// TIA Portal V20 export
// export: Created 2025-12-01T14:57:27.0785066Z, ExportSetting None, DisplayName Totally Integrated Automation Portal, DisplayVersion V20 Update 3, DisplayName TIA Portal Openness, DisplayVersion V20 Update 3, DisplayName TIA Portal Version Control Interface, DisplayVersion V20 Update 3, DisplayName STEP 7 Professional, DisplayVersion V20 Update 3, DisplayName STEP 7 Safety, DisplayVersion V20 Update 2, DisplayName WinCC Basic/Comfort/Advanced, DisplayVersion V20 Update 3, DisplayName WinCC Professional, DisplayVersion V20 Update 3, DisplayName WinCC Unified, DisplayVersion V20 Update 3
FUNCTION_BLOCK "FB609_RepartoEntradas_2E_Quimarox"   // FB609, LAD
{ S7_Optimized_Access := 'FALSE' }
// stored: AutoNumber false, SetENOAutomatically false
   VAR_INPUT
      Mesa_E1 : UInt;
      Mesa_E2 : UInt;
      AVTF_ME1_MSig : Bool;
      AVTF_ME2_MSig : Bool;
      V_Reparto_ME1 : UInt;
      V_Reparto_ME2 : UInt;
   END_VAR
   VAR_OUTPUT
      Permiso_ME1_MSig : Bool;
      Permiso_ME2_MSig : Bool;
   END_VAR
   VAR
      CNT_Entradas_ME1 : UInt;
      CNT_Entradas_ME2 : UInt;
      MFP_Entrada_ME1 : Bool;
      MFP_Entrada_ME2 : Bool;
      MEntrando_ME1 : Bool;
      MEntrando_ME2 : Bool;
   END_VAR
   VAR_TEMP   // added for the SCL form of the ladder/FBD networks
      _w1 : Bool;
   END_VAR
BEGIN

REGION Network 1: >>>>>>>> INICIALIZAR
END_REGION

REGION Network 2: >>>>>>>> CONTROL DE LOS CONTADORES DE LAS ENTRADAS
END_REGION

REGION Network 3: Numero de Entradas realizadas desde ME1 (Contador)
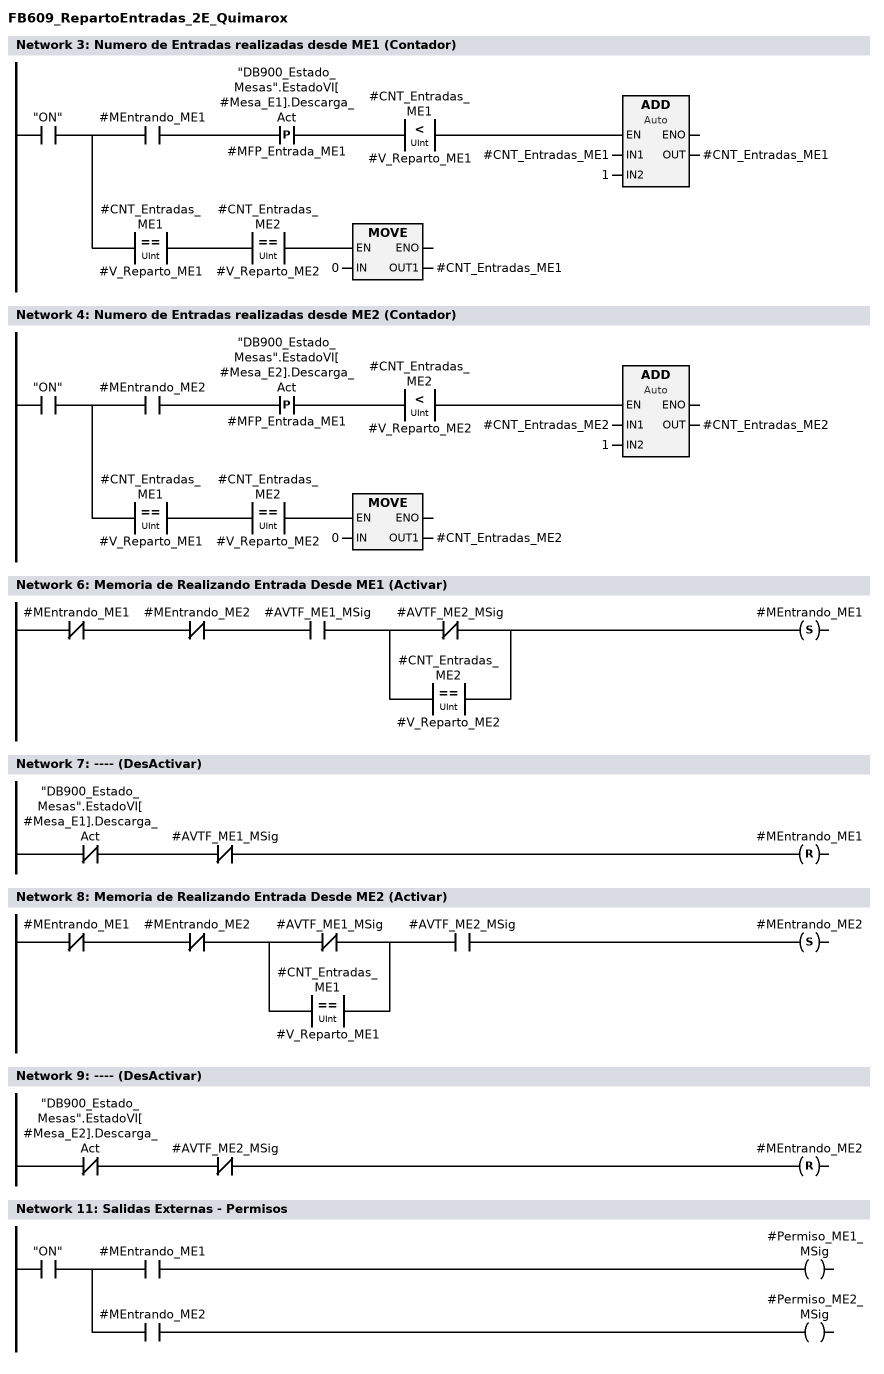
   RUNG wire#powerrail
      Contact( "ON" )
      wire#w1
      Contact( #MEntrando_ME1 )
      P_Contact(operand := "DB900_Estado_Mesas".EstadoVI[#Mesa_E1].Descarga_Act, bit := #MFP_Entrada_ME1)
      { S7_Templates := "SrcType := UInt" } LT_Contact(in1 := #CNT_Entradas_ME1, in2 := #V_Reparto_ME1)
      Add(in1 := #CNT_Entradas_ME1, in2 := 1, out => #CNT_Entradas_ME1)
   END_RUNG
   RUNG wire#w1
      { S7_Templates := "SrcType := UInt" } EQ_Contact(in1 := #CNT_Entradas_ME1, in2 := #V_Reparto_ME1)
      { S7_Templates := "SrcType := UInt" } EQ_Contact(in1 := #CNT_Entradas_ME2, in2 := #V_Reparto_ME2)
      Move(in := 0, out1 => #CNT_Entradas_ME1)
   END_RUNG
   // the same network as SCL:
   #_w1 := "ON" AND #MEntrando_ME1 AND "DB900_Estado_Mesas".EstadoVI[#Mesa_E1].Descarga_Act AND NOT #MFP_Entrada_ME1;   // rising edge of "DB900_Estado_Mesas".EstadoVI[#Mesa_E1].Descarga_Act
   #MFP_Entrada_ME1 := "DB900_Estado_Mesas".EstadoVI[#Mesa_E1].Descarga_Act;
   IF #_w1 AND (#CNT_Entradas_ME1 < #V_Reparto_ME1) THEN #CNT_Entradas_ME1 := #CNT_Entradas_ME1 + 1; END_IF;
   IF "ON" AND (#CNT_Entradas_ME1 = #V_Reparto_ME1) AND (#CNT_Entradas_ME2 = #V_Reparto_ME2) THEN
       #CNT_Entradas_ME1 := 0;
   END_IF;
END_REGION

REGION Network 4: Numero de Entradas realizadas desde ME2 (Contador)
   RUNG wire#powerrail
      Contact( "ON" )
      wire#w1
      Contact( #MEntrando_ME2 )
      P_Contact(operand := "DB900_Estado_Mesas".EstadoVI[#Mesa_E2].Descarga_Act, bit := #MFP_Entrada_ME1)
      { S7_Templates := "SrcType := UInt" } LT_Contact(in1 := #CNT_Entradas_ME2, in2 := #V_Reparto_ME2)
      Add(in1 := #CNT_Entradas_ME2, in2 := 1, out => #CNT_Entradas_ME2)
   END_RUNG
   RUNG wire#w1
      { S7_Templates := "SrcType := UInt" } EQ_Contact(in1 := #CNT_Entradas_ME1, in2 := #V_Reparto_ME1)
      { S7_Templates := "SrcType := UInt" } EQ_Contact(in1 := #CNT_Entradas_ME2, in2 := #V_Reparto_ME2)
      Move(in := 0, out1 => #CNT_Entradas_ME2)
   END_RUNG
   // the same network as SCL:
   #_w1 := "ON" AND #MEntrando_ME2 AND "DB900_Estado_Mesas".EstadoVI[#Mesa_E2].Descarga_Act AND NOT #MFP_Entrada_ME1;   // rising edge of "DB900_Estado_Mesas".EstadoVI[#Mesa_E2].Descarga_Act
   #MFP_Entrada_ME1 := "DB900_Estado_Mesas".EstadoVI[#Mesa_E2].Descarga_Act;
   IF #_w1 AND (#CNT_Entradas_ME2 < #V_Reparto_ME2) THEN #CNT_Entradas_ME2 := #CNT_Entradas_ME2 + 1; END_IF;
   IF "ON" AND (#CNT_Entradas_ME1 = #V_Reparto_ME1) AND (#CNT_Entradas_ME2 = #V_Reparto_ME2) THEN
       #CNT_Entradas_ME2 := 0;
   END_IF;
END_REGION

REGION Network 5: >>>>>>>> MEMORIA DE ESTADO - ENTRANDO
END_REGION

REGION Network 6: Memoria de Realizando Entrada Desde ME1 (Activar)
   RUNG wire#powerrail
      I_Contact( #MEntrando_ME1 )
      I_Contact( #MEntrando_ME2 )
      Contact( #AVTF_ME1_MSig )
      wire#w1
      I_Contact( #AVTF_ME2_MSig )
      wire#w2
      S_Coil( #MEntrando_ME1 )
   END_RUNG
   RUNG wire#w1
      { S7_Templates := "SrcType := UInt" } EQ_Contact(in1 := #CNT_Entradas_ME2, in2 := #V_Reparto_ME2)
   END_RUNG wire#w2
   // the same network as SCL:
   IF NOT #MEntrando_ME1 AND NOT #MEntrando_ME2 AND #AVTF_ME1_MSig AND (NOT #AVTF_ME2_MSig OR (#CNT_Entradas_ME2 = #V_Reparto_ME2)) THEN
       #MEntrando_ME1 := TRUE;
   END_IF;
END_REGION

REGION Network 7: ---- (DesActivar)
   RUNG wire#powerrail
      I_Contact( "DB900_Estado_Mesas".EstadoVI[#Mesa_E1].Descarga_Act )
      I_Contact( #AVTF_ME1_MSig )
      R_Coil( #MEntrando_ME1 )
   END_RUNG
   // the same network as SCL:
   IF NOT "DB900_Estado_Mesas".EstadoVI[#Mesa_E1].Descarga_Act AND NOT #AVTF_ME1_MSig THEN
       #MEntrando_ME1 := FALSE;
   END_IF;
END_REGION

REGION Network 8: Memoria de Realizando Entrada Desde ME2 (Activar)
   RUNG wire#powerrail
      I_Contact( #MEntrando_ME1 )
      I_Contact( #MEntrando_ME2 )
      wire#w1
      I_Contact( #AVTF_ME1_MSig )
      wire#w2
      Contact( #AVTF_ME2_MSig )
      S_Coil( #MEntrando_ME2 )
   END_RUNG
   RUNG wire#w1
      { S7_Templates := "SrcType := UInt" } EQ_Contact(in1 := #CNT_Entradas_ME1, in2 := #V_Reparto_ME1)
   END_RUNG wire#w2
   // the same network as SCL:
   IF NOT #MEntrando_ME1 AND NOT #MEntrando_ME2 AND (NOT #AVTF_ME1_MSig OR (#CNT_Entradas_ME1 = #V_Reparto_ME1)) AND #AVTF_ME2_MSig THEN
       #MEntrando_ME2 := TRUE;
   END_IF;
END_REGION

REGION Network 9: ---- (DesActivar)
   RUNG wire#powerrail
      I_Contact( "DB900_Estado_Mesas".EstadoVI[#Mesa_E2].Descarga_Act )
      I_Contact( #AVTF_ME2_MSig )
      R_Coil( #MEntrando_ME2 )
   END_RUNG
   // the same network as SCL:
   IF NOT "DB900_Estado_Mesas".EstadoVI[#Mesa_E2].Descarga_Act AND NOT #AVTF_ME2_MSig THEN
       #MEntrando_ME2 := FALSE;
   END_IF;
END_REGION

REGION Network 10: >>>>>>>> ACTIVACION DE SALIDAS
END_REGION

REGION Network 11: Salidas Externas - Permisos
   RUNG wire#powerrail
      Contact( "ON" )
      wire#w1
      Contact( #MEntrando_ME1 )
      Coil( #Permiso_ME1_MSig )
   END_RUNG
   RUNG wire#w1
      Contact( #MEntrando_ME2 )
      Coil( #Permiso_ME2_MSig )
   END_RUNG
   // the same network as SCL:
   #Permiso_ME1_MSig := "ON" AND #MEntrando_ME1;
   #Permiso_ME2_MSig := "ON" AND #MEntrando_ME2;
END_REGION
END_FUNCTION_BLOCK
